INTERFACE ITF_BaseLoggerElement_HMI_Connector

METHOD PUBLIC GetCode : STRING
VAR_INPUT
END_VAR
END_METHOD

METHOD PUBLIC GetID : UINT
VAR_INPUT
END_VAR
END_METHOD

METHOD PUBLIC GetIdentyfier : ST_BaseElementIdentifier
VAR_INPUT
END_VAR
END_METHOD

METHOD PUBLIC GetName : ST_BaseLabel
VAR_INPUT
END_VAR
END_METHOD

METHOD PUBLIC GetType : E_BaseElementType
VAR_INPUT
END_VAR
END_METHOD

END_INTERFACE

(* stored: Version 1.1.0.1
   Itf ITF_BaseLoggerElement_HMI_Connector: Id {18066f33-5cce-0b8b-2b60-e60e4addcc02}
   Method GetCode: Id {f5cf3e5c-088f-0e43-06f5-119997559e59}
   Method GetID: Id {6d80811c-c1cb-062f-0769-541a69ee6d76}
   Method GetIdentyfier: Id {ac6e2f1d-ef73-047b-0178-a3d1abb02eb3}
   Method GetName: Id {8b277639-3747-0d1b-09fd-1b4180f8280b}
   Method GetType: Id {39784064-3fc4-0e64-092d-21b915a721a1} *)
